FUNCTION_BLOCK FB_NOTT_STEPPER_SHUTTER EXTENDS FB_MOTOR
VAR_INPUT
END_VAR
VAR_OUTPUT
END_VAR
VAR
END_VAR


SUPER^();

END_FUNCTION_BLOCK

(* stored: Version 1.1.0.1, ProductVersion 3.1.4024.14
   POU FB_NOTT_STEPPER_SHUTTER: Id {2b5f4452-810d-4eb6-9497-660721820ccc}, SpecialFunc None *)
